FUNCTION_BLOCK vishalTest
VAR_INPUT
END_VAR
VAR_OUTPUT
END_VAR
VAR
END_VAR

END_FUNCTION_BLOCK

(* stored: Version 1.1.0.1, ProductVersion 3.1.4024.16
   POU vishalTest: Id {36e926be-3fb1-41ad-8761-5d2f09e882c5}, SpecialFunc None *)
